{attribute 'qualified_only'}
{attribute 'strict'}
{attribute 'to_string'}
TYPE E_MotorZuigSchuifStatus :
(
	Kort := 0,
	Lang,
	GoToKort,
	GoToLang,
	Error
);
END_TYPE

(* stored: Version 1.1.0.1
   DUT E_MotorZuigSchuifStatus: Id {664bc50d-fe32-40a6-aa94-9e04edd3a8d8} *)
